(* CODESYS project GardenWatering.project
   Title: Garden Watering
   Version: 1.0
   Company: TK Automation
   Author: Toni Kucic

Project tree, tasks and I/O mapping:
  SoftPLC : CODESYS Control Win V3 x64, 3S - Smart Software Solutions GmbH, version 3.5.12.0
    application Application
      libraries: Standard, * (System); TkAutomationLib, 1.0 (TkAutomation); Util, * (System); Standard64, * (System); VisuDialogs, * (System)
      task VISU_TASK (cyclic, interval 50 ms, priority 31) calls VisuElems.Visu_Prg
      task xsim02 (cyclic, interval t#20ms, priority 2) calls xsim02
      task xc02_Task (cyclic, interval t#20ms, priority 1) calls xc02_GardenWatering, xc02_GardenWatering_Encoder
      FunctionalDescriptions/
        FD_GardenWatering
      image pool ImagePool
      FunctionBLocks/
        function block Servo [ST]
      IO/
        global variables xgv02
        Symbols
      Control/
        program xc02_GardenWatering [ST]
        program xc02_GardenWatering_Encoder [ST]
      Simulator/
        program xsim02 [ST]
      HMI/
        visualisation xv02_GardenWatering
  libraries: VisuSymbols, 3.5.10.0 (System)
  00000000-0000-0000-0000-000000000000|C:\Users\Toni\Google Drive\Projekti\PLC projekti\tkautomation school\Functional Descriptions\FD_GardenWatering.docx
  text list GlobalTextList
  5ce3da45-db07-42e7-a21c-a00fff4ed8f6|Car1.png
  5ce3da45-db07-42e7-a21c-a00fff4ed8f6|Projects\breaker1.jpg
  5ce3da45-db07-42e7-a21c-a00fff4ed8f6|Projects\breaker2.jpg
  5ce3da45-db07-42e7-a21c-a00fff4ed8f6|Projects\Ventilator1.jpg
  5ce3da45-db07-42e7-a21c-a00fff4ed8f6|Projects\Ventilator2.jpg
  5ce3da45-db07-42e7-a21c-a00fff4ed8f6|Projects\main-switchboard_1.jpg
  5ce3da45-db07-42e7-a21c-a00fff4ed8f6|Projects\breaker1.jpg
  5ce3da45-db07-42e7-a21c-a00fff4ed8f6|Projects\breaker2.jpg
  5ce3da45-db07-42e7-a21c-a00fff4ed8f6|Projects\cloud with rain.jpg
  5ce3da45-db07-42e7-a21c-a00fff4ed8f6|Car2.png
  text list System
  5ce3da45-db07-42e7-a21c-a00fff4ed8f6|Car3.png
  5ce3da45-db07-42e7-a21c-a00fff4ed8f6|Projects\Ventilator1small.jpg
  5ce3da45-db07-42e7-a21c-a00fff4ed8f6|Projects\Ventilator2small.jpg
  5ce3da45-db07-42e7-a21c-a00fff4ed8f6|Projects\igrasatasterima.JPG
  5ce3da45-db07-42e7-a21c-a00fff4ed8f6|Projects\empty-road-intersection-icon-cartoon-style-H67GFG.jpg
  5ce3da45-db07-42e7-a21c-a00fff4ed8f6|Projects\traffic_light_05.jpgsmall.jpg
  5ce3da45-db07-42e7-a21c-a00fff4ed8f6|Projects\breaker1.jpg
  5ce3da45-db07-42e7-a21c-a00fff4ed8f6|Projects\breaker2.jpg
  5ce3da45-db07-42e7-a21c-a00fff4ed8f6|C:\Users\Toni\Google Drive\Projekti\PLC projekti\Materijali\traffic_light_05.jpgsmall.jpg
  5ce3da45-db07-42e7-a21c-a00fff4ed8f6|boom.png
  5ce3da45-db07-42e7-a21c-a00fff4ed8f6|bottle_empty.png
  5ce3da45-db07-42e7-a21c-a00fff4ed8f6|bottle_broken.png
  5ce3da45-db07-42e7-a21c-a00fff4ed8f6|bottle_halffull.png
  5ce3da45-db07-42e7-a21c-a00fff4ed8f6|bottle_full.png
  5ce3da45-db07-42e7-a21c-a00fff4ed8f6|roller1.png
  5ce3da45-db07-42e7-a21c-a00fff4ed8f6|roller2.png
  5ce3da45-db07-42e7-a21c-a00fff4ed8f6|cranebackground.png
  5ce3da45-db07-42e7-a21c-a00fff4ed8f6|cranemover.png
  5ce3da45-db07-42e7-a21c-a00fff4ed8f6|hook.png
  5ce3da45-db07-42e7-a21c-a00fff4ed8f6|trafficlightsystem.jpg
  5ce3da45-db07-42e7-a21c-a00fff4ed8f6|Car4.png
*)

// SoftPLC/Application/IO/xgv02
{attribute 'qualified_only'}
VAR_GLOBAL
	
	//Configuration

	//Inputs
	HorizontalS1 : BOOL;
	HorizontalS2 : BOOL;
	VerticalS1 : BOOL;
	VerticalS2 : BOOL;
	
	//Data from encoder
	PositionX : REAL;
	PositionY : REAL;
	
	(* HMI *)
	HMIUp : BOOL;
	HMIDown : BOOL;
	HMIRight : BOOL;
	HMILeft : BOOL;
	HMIUpRight : BOOL;
	HMIUpLeft : BOOL;
	HMIDownRight : BOOL;
	HMIDownLeft : BOOL;
	HMICoorXCmd : REAL;
	HMICoorYCmd : REAL;
	HMIOpenWater : BOOL;
	Remote : BOOL;
	Reset : BOOL;
	
	//Outputs
	HorizontalRight : BOOL;
	HorizontalLeft : BOOL;
	VerticalUp: BOOL;
	VerticalDown : BOOL;
	OpenWaterValve : BOOL;
END_VAR

// SoftPLC/Application/Simulator/xsim02
PROGRAM xsim02
VAR
	CollisionDetector: CollisionDetection;
	FlowerDeathTimer: TON;
	vResetSIM: BOOL;
	vFlowers : ARRAY [0..59] OF DWORD := [60(16#FF73B98B)];
	i : INT;
vFlowersXY : ARRAY [0..59, 0..1] OF INT := [276,253,	381,253,	486,253,	591,253,	696,253,	801,253,	906,253,	1011,253,	1116,253,	1221,253,
												276,354,	381,354,	486,354,	591,354,	696,354,	801,354,	906,354,	1011,354,	1116,354,	1221,354,
												276,455,	381,455,	486,455,	591,455,	696,455,	801,455,	906,455,	1011,455,	1116,455,	1221,455,
												276,556,	381,556,	486,556,	591,556,	696,556,	801,556,	906,556,	1011,556,	1116,556,	1221,556,
												276,667,	381,667,	486,667,	591,667,	696,667,	801,667,	906,667,	1011,667,	1116,667,	1221,667,
												276,768,	381,768,	486,768,	591,768,	696,768,	801,768,	906,768,	1011,768,	1116,768,	1221,768]; (* Coordinates of flowers in format Flower0 -x,y *)

END_VAR

(* If the plaform covers the flower it will reset its color to initial *)
FOR i:=0 TO 59 BY 1 DO
	CollisionDetector(
		xcor1:= xgv02.PositionX, 
		ycor1:= xgv02.PositionY, 
		height1:= 10, 
		width1:= 10, 
		xcor2:= vFlowersXY[i,0], 
		ycor2:= vFlowersXY[i,1], 
		height2:= 70 , 
		width2:= 70);
	IF CollisionDetector.isCollision AND xgv02.OpenWaterValve THEN
		vFlowers[i] := 16#FF73B98B;
	END_IF
END_FOR

FlowerDeathTimer(IN:=TRUE, PT:=T#60S);
(* Flowers fade its color *)
IF FlowerDeathTimer.Q THEN
	FOR i:=0 TO 59 BY 1 DO
		IF vFlowers[i] > 16#0073B98B THEN
			vFlowers[i] := vFlowers[i] - 16#01000000;
		END_IF;
	END_FOR
	FlowerDeathTimer.IN := FALSE;
END_IF;

END_PROGRAM

// SoftPLC/Application/Control/xc02_GardenWatering
PROGRAM xc02_GardenWatering
VAR
	vFlowersXY : ARRAY [0..59, 0..1] OF INT := [276,253,	381,253,	486,253,	591,253,	696,253,	801,253,	906,253,	1011,253,	1116,253,	1221,253,
												276,354,	381,354,	486,354,	591,354,	696,354,	801,354,	906,354,	1011,354,	1116,354,	1221,354,
												276,455,	381,455,	486,455,	591,455,	696,455,	801,455,	906,455,	1011,455,	1116,455,	1221,455,
												276,556,	381,556,	486,556,	591,556,	696,556,	801,556,	906,556,	1011,556,	1116,556,	1221,556,
												276,667,	381,667,	486,667,	591,667,	696,667,	801,667,	906,667,	1011,667,	1116,667,	1221,667,
												276,768,	381,768,	486,768,	591,768,	696,768,	801,768,	906,768,	1011,768,	1116,768,	1221,768]; (* Coordinates of flowers in format Flower0 -x,y *)

	vManual: BOOL;
	vXCMD : REAL;
	vYCMD : REAL;
	i: INT;
	Watering: TON;
	ActuatorOverFlower : CollisionDetection;
END_VAR

(* Control from the graphics *)
IF NOT xgv02.Remote THEN
	xgv02.HorizontalLeft := xgv02.HMIDownLeft OR xgv02.HMILeft OR xgv02.HMIUpLeft;
	xgv02.HorizontalRight := xgv02.HMIDownRight OR xgv02.HMIRight OR xgv02.HMIUpRight;
	xgv02.VerticalUp := xgv02.HMIUpLeft OR xgv02.HMIUp OR xgv02.HMIUpRight;
	xgv02.VerticalDown := xgv02.HMIDownLeft OR xgv02.HMIDown OR xgv02.HMIDownRight;
	xgv02.OpenWaterValve := xgv02.HMIOpenWater;
END_IF;

(* Coordinate control *)
IF xgv02.Remote AND vManual THEN
	vXCMD := xgv02.HMICoorXCmd;
	vYCMD := xgv02.HMICoorYCmd;
ELSE
	xgv02.HMICoorXCmd := xgv02.PositionX;
	xgv02.HMICoorYCmd := xgv02.PositionY;
END_IF

(* Full automatic algorithm *)
IF xgv02.Remote AND NOT vManual THEN
	vXCMD := vFlowersXY[i,0]+ 30;
	vYCMD := vFlowersXY[i,1]+ 30;
	
	ActuatorOverFlower(
		xcor1:= xgv02.PositionX, 
		ycor1:= xgv02.PositionY, 
		height1:= 10, 
		width1:= 10, 
		xcor2:= vFlowersXY[i,0], 
		ycor2:= vFlowersXY[i,1], 
		height2:= 70, 
		width2:= 70);
		
	IF 	ActuatorOverFlower.isCollision THEN
		Watering(IN:=TRUE, PT:=T#3S);
		xgv02.OpenWaterValve := TRUE;
	END_IF;
	IF ActuatorOverFlower.isCollision AND Watering.Q THEN
		Watering(IN := FALSE);
		xgv02.OpenWaterValve:= FALSE;
		i:= i + 1;	
	END_IF
END_IF
IF i = 59 THEN
	i := 0;
END_IF

(* Actual motor movement section *)
IF xgv02.Remote THEN
	IF vXCMD > xgv02.PositionX - 2 THEN
		xgv02.HorizontalLeft := FALSE;
		xgv02.HorizontalRight := TRUE;
	ELSIF vXCMD < xgv02.PositionX + 2 THEN
		xgv02.HorizontalLeft := TRUE;
		xgv02.HorizontalRight := FALSE;
	ELSE
		xgv02.HorizontalLeft := FALSE;
		xgv02.HorizontalRight := FALSE;
	END_IF;
	
	IF vYCMD < xgv02.PositionY - 2THEN
		xgv02.VerticalUp := TRUE;
		xgv02.VerticalDown := FALSE;
	ELSIF vYCMD > xgv02.PositionY + 2 THEN
		xgv02.VerticalUp := FALSE;
		xgv02.VerticalDown := TRUE;
	ELSE
		xgv02.VerticalUp := FALSE;
		xgv02.VerticalDown := FALSE;
	END_IF;
END_IF;

END_PROGRAM

// SoftPLC/Application/Control/xc02_GardenWatering_Encoder
PROGRAM xc02_GardenWatering_Encoder
VAR
	HorizontalAxis: Servo;
	VerticalAxis: Servo;
	rtHIncrement : R_TRIG;
	rtHDecrement : R_TRIG;
	rtVIncrement : R_TRIG;
	rtVDecrement : R_TRIG;
	vHorizontalS1Old: BOOL;
	vHorizontalS2Old: BOOL;
	vVerticalS1Old: BOOL;
	vVerticalS2Old: BOOL;
	PositionCounterVerticalAxis: CTUD;
	vHorizontalPos: DINT;
	PositionCounterHorizontalAxis: CTUD;
	vVerticalPos: WORD;
	vPositionX: REAL;
	vPositionY: REAL;
	vHorizontalLimit: BOOL;
	vVerticalLimit: BOOL;
	vPlatformActualPosX : REAL;
	vPlatformActualPosY : REAL;
END_VAR

(* The actual servos that move the watering equipment *)
vHorizontalLimit := (vPositionX >= 940 AND NOT xgv02.HorizontalLeft)
				  OR (vPositionX <= 0 AND NOT xgv02.HorizontalRight);
vVerticalLimit := (vPositionY >= 500 AND NOT xgv02.VerticalUp)
			    OR (vPositionY <= 0 AND NOT xgv02.VerticalDown);

(* Maximum range - 940 steps *)
HorizontalAxis(
	CmdFwd:= xgv02.HorizontalRight AND NOT vHorizontalLimit, 
	CmdRev:= xgv02.HorizontalLeft AND NOT vHorizontalLimit, 
	PulseWidth:= T#0.1S , 
	S1=> xgv02.HorizontalS1, 
	S2=> xgv02.HorizontalS2);
	
(* Maximum range - 500 steps *)	
VerticalAxis(
	CmdFwd:= xgv02.VerticalDown AND NOT vVerticalLimit, 
	CmdRev:= xgv02.VerticalUp AND NOT vVerticalLimit, 
	PulseWidth:= T#0.1S , 
	S1=> xgv02.VerticalS1, 
	S2=> xgv02.VerticalS2);

IF xgv02.HorizontalS1 <> vHorizontalS1Old THEN
	IF xgv02.HorizontalS1 <> xgv02.HorizontalS2 THEN
		rtHIncrement(CLK:=TRUE);
	ELSE
		rtHDecrement(CLK:=TRUE);
	END_IF
ELSE
	rtHIncrement(CLK:=FALSE);
	rtHDecrement(CLK:=FALSE);
END_IF

IF xgv02.VerticalS1 <> vVerticalS1Old THEN
	IF xgv02.VerticalS1 <> xgv02.VerticalS2 THEN
		rtVIncrement(CLK:=TRUE);
	ELSE
		rtVDecrement(CLK:=TRUE);
	END_IF
ELSE
	rtVIncrement(CLK:=FALSE);
	rtVDecrement(CLK:=FALSE);
END_IF

PositionCounterHorizontalAxis(
	CU:= rtHIncrement.Q, 
	CD:= rtHDecrement.Q, 
	CV=> vHorizontalPos);

PositionCounterVerticalAxis(
	CU:= rtVIncrement.Q, 
	CD:= rtVDecrement.Q, 
	CV=> vVerticalPos);
	
(* Position of the system in the graphics*)
(* For every 1 pulses we move 5 px *)
vPositionX := (DINT_TO_REAL(vHorizontalPos)/ 1) * 5;
vPositionY := (DINT_TO_REAL(vVerticalPos)/ 1) * 5;
	
vHorizontalS1Old := xgv02.HorizontalS1;
vVerticalS1Old := xgv02.VerticalS1;
(* This is to counter the starting offset in the graphics *)
vPlatformActualPosX := 307 + vPositionX;
vPlatformActualPosY := 279 + vPositionY;

(* Send the platform position to other programs *)
xgv02.PositionX := vPlatformActualPosX;
xgv02.PositionY := vPlatformActualPosY;

END_PROGRAM

// SoftPLC/Application/FunctionBLocks/Servo
FUNCTION_BLOCK Servo
VAR_INPUT
	CmdFwd : BOOL := FALSE;
	CmdRev : BOOL := FALSE;
	PulseWidth : TIME := T#0.1S; (* Width of a pulse from the hall effect sensor when its above magnetic surface *)
END_VAR
VAR_OUTPUT
	S1 : BOOL := FALSE;
	S2 : BOOL := FALSE;
END_VAR
VAR
	tofS2 : TOF;
	tonS2 : TON;
	blink : BLINK;
	blinkOld: BOOL;
	vStartBlinker: BOOL;
END_VAR

vStartBlinker := (CmdFwd OR CmdRev) AND NOT (CmdFwd AND CmdRev);
Blink(ENABLE := vStartBlinker, TIMELOW:= PulseWidth, TIMEHIGH := PulseWidth);

tonS2(IN := blink.OUT, PT:=PulseWidth/2);
tofS2(IN := NOT tonS2.Q AND blinkOld, PT:=PulseWidth/2);
 
blinkOld := tonS2.Q;

IF CmdFwd THEN
	S1 := blink.OUT;
	S2 := tonS2.Q OR tofS2.Q;
ELSIF CmdRev THEN
	S1 := tonS2.Q OR tofS2.Q;
	S2 := blink.OUT;
END_IF

END_FUNCTION_BLOCK

// SoftPLC/Application/HMI/xv02_GardenWatering
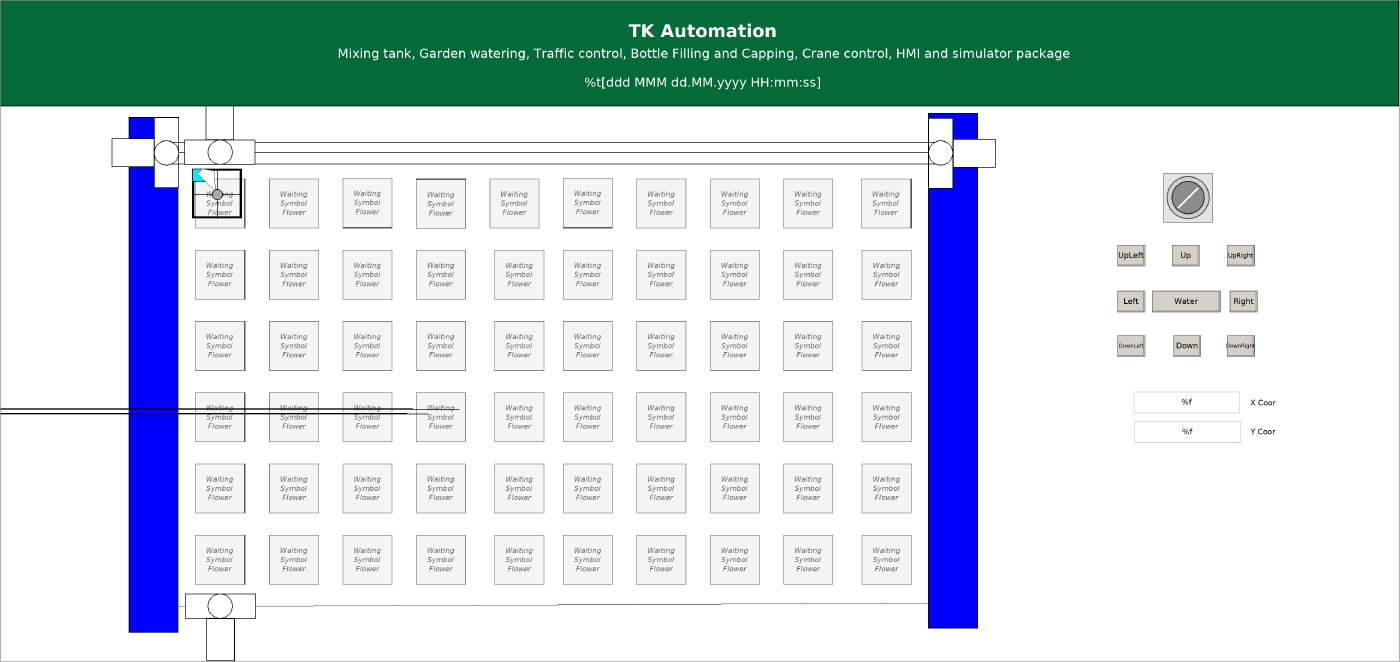
VISUALIZATION xv02_GardenWatering  // 1982x938
    RoundedRectangle (381,354 70x70), colour variable: xsim02.vFlowers[11]
    RoundedRectangle (485,354 70x70), colour variable: xsim02.vFlowers[12]
    RoundedRectangle (589,354 70x70), colour variable: xsim02.vFlowers[13]
    RoundedRectangle (700,354 70x70), colour variable: xsim02.vFlowers[14]
    RoundedRectangle (797,354 70x70), colour variable: xsim02.vFlowers[15]
    RoundedRectangle (901,354 70x70), colour variable: xsim02.vFlowers[16]
    RoundedRectangle (1005,354 70x70), colour variable: xsim02.vFlowers[17]
    RoundedRectangle (1109,354 70x70), colour variable: xsim02.vFlowers[18]
    RoundedRectangle (1220,354 70x70), colour variable: xsim02.vFlowers[19]
    RoundedRectangle (381,455 70x70), colour variable: xsim02.vFlowers[21]
    RoundedRectangle (485,455 70x70), colour variable: xsim02.vFlowers[22]
    RoundedRectangle (589,455 70x70), colour variable: xsim02.vFlowers[23]
    RoundedRectangle (700,455 70x70), colour variable: xsim02.vFlowers[24]
    RoundedRectangle (797,455 70x70), colour variable: xsim02.vFlowers[25]
    RoundedRectangle (901,455 70x70), colour variable: xsim02.vFlowers[26]
    RoundedRectangle (1005,455 70x70), colour variable: xsim02.vFlowers[27]
    RoundedRectangle (1109,455 70x70), colour variable: xsim02.vFlowers[28]
    RoundedRectangle (1220,455 70x70), colour variable: xsim02.vFlowers[29]
    RoundedRectangle (381,556 70x70), colour variable: xsim02.vFlowers[31]
    RoundedRectangle (485,556 70x70), colour variable: xsim02.vFlowers[32]
    RoundedRectangle (589,556 70x70), colour variable: xsim02.vFlowers[33]
    RoundedRectangle (700,556 70x70), colour variable: xsim02.vFlowers[34]
    RoundedRectangle (797,556 70x70), colour variable: xsim02.vFlowers[35]
    RoundedRectangle (901,556 70x70), colour variable: xsim02.vFlowers[36]
    RoundedRectangle (1005,556 70x70), colour variable: xsim02.vFlowers[37]
    RoundedRectangle (1109,556 70x70), colour variable: xsim02.vFlowers[38]
    RoundedRectangle (1220,556 70x70), colour variable: xsim02.vFlowers[39]
    RoundedRectangle (381,657 70x70), colour variable: xsim02.vFlowers[41]
    RoundedRectangle (485,657 70x70), colour variable: xsim02.vFlowers[42]
    RoundedRectangle (589,657 70x70), colour variable: xsim02.vFlowers[43]
    RoundedRectangle (700,657 70x70), colour variable: xsim02.vFlowers[44]
    RoundedRectangle (797,657 70x70), colour variable: xsim02.vFlowers[45]
    RoundedRectangle (901,657 70x70), colour variable: xsim02.vFlowers[46]
    RoundedRectangle (1005,657 70x70), colour variable: xsim02.vFlowers[47]
    RoundedRectangle (1109,657 70x70), colour variable: xsim02.vFlowers[48]
    RoundedRectangle (1220,657 70x70), colour variable: xsim02.vFlowers[49]
    RoundedRectangle (381,758 70x70), colour variable: xsim02.vFlowers[51]
    RoundedRectangle (485,758 70x70), colour variable: xsim02.vFlowers[52]
    RoundedRectangle (589,758 70x70), colour variable: xsim02.vFlowers[53]
    RoundedRectangle (700,758 70x70), colour variable: xsim02.vFlowers[54]
    RoundedRectangle (797,758 70x70), colour variable: xsim02.vFlowers[55]
    RoundedRectangle (901,758 70x70), colour variable: xsim02.vFlowers[56]
    RoundedRectangle (1005,758 70x70), colour variable: xsim02.vFlowers[57]
    RoundedRectangle (1109,758 70x70), colour variable: xsim02.vFlowers[58]
    RoundedRectangle (1220,758 70x70), colour variable: xsim02.vFlowers[59]
    Group (276,253 71x70)
        RoundedRectangle (1,0 70x70), colour variable: xsim02.vFlowers[0]
        WaitingSymbolFlower (0,0 70x70)
    Group (276,354 71x70)
        RoundedRectangle (1,0 70x70), colour variable: xsim02.vFlowers[10]
        WaitingSymbolFlower (0,0 70x70)
    Group (276,455 71x70)
        RoundedRectangle (1,0 70x70), colour variable: xsim02.vFlowers[20]
        WaitingSymbolFlower (0,0 70x70)
    Group (276,758 71x70)
        RoundedRectangle (1,0 70x70), colour variable: xsim02.vFlowers[50]
        WaitingSymbolFlower (0,0 70x70)
    Group (276,556 71x70)
        RoundedRectangle (1,0 70x70), colour variable: xsim02.vFlowers[30]
        WaitingSymbolFlower (0,0 70x70)
    Group (276,657 71x70)
        RoundedRectangle (1,0 70x70), colour variable: xsim02.vFlowers[40]
        WaitingSymbolFlower (0,0 70x70)
    Group (381,253 70x70)
        RoundedRectangle (0,0 70x70), colour variable: xsim02.vFlowers[1]
        WaitingSymbolFlower (0,0 70x70)
    WaitingSymbolFlower (381,354 70x70)
    WaitingSymbolFlower (381,455 70x70)
    WaitingSymbolFlower (381,758 70x70)
    WaitingSymbolFlower (381,556 70x70)
    WaitingSymbolFlower (381,657 70x70)
    Group (589,253 70x71)
        RoundedRectangle (0,0 70x70), colour variable: xsim02.vFlowers[2]
        WaitingSymbolFlower (0,1 70x70)
    WaitingSymbolFlower (485,354 70x70)
    WaitingSymbolFlower (485,455 70x70)
    WaitingSymbolFlower (485,758 70x70)
    WaitingSymbolFlower (485,556 70x70)
    WaitingSymbolFlower (485,657 70x70)
    Group (485,252 70x71)
        RoundedRectangle (0,1 70x70), colour variable: xsim02.vFlowers[3]
        WaitingSymbolFlower (0,0 70x70)
    WaitingSymbolFlower (589,354 70x70)
    WaitingSymbolFlower (589,455 70x70)
    WaitingSymbolFlower (589,758 70x70)
    WaitingSymbolFlower (589,556 70x70)
    WaitingSymbolFlower (589,657 70x70)
    Group (693,253 70x70)
        RoundedRectangle (0,0 70x70), colour variable: xsim02.vFlowers[4]
        WaitingSymbolFlower (0,0 70x70)
    WaitingSymbolFlower (700,354 70x70)
    WaitingSymbolFlower (700,455 70x70)
    WaitingSymbolFlower (700,758 70x70)
    WaitingSymbolFlower (700,556 70x70)
    WaitingSymbolFlower (700,657 70x70)
    Group (797,252 70x71)
        RoundedRectangle (0,1 70x70), colour variable: xsim02.vFlowers[5]
        WaitingSymbolFlower (0,0 70x70)
    WaitingSymbolFlower (797,354 70x70)
    WaitingSymbolFlower (797,455 70x70)
    WaitingSymbolFlower (797,758 70x70)
    WaitingSymbolFlower (797,556 70x70)
    WaitingSymbolFlower (797,657 70x70)
    Group (901,253 70x70)
        RoundedRectangle (0,0 70x70), colour variable: xsim02.vFlowers[6]
        WaitingSymbolFlower (0,0 70x70)
    WaitingSymbolFlower (901,354 70x70)
    WaitingSymbolFlower (901,455 70x70)
    WaitingSymbolFlower (901,758 70x70)
    WaitingSymbolFlower (901,556 70x70)
    WaitingSymbolFlower (901,657 70x70)
    Group (1005,253 70x70)
        RoundedRectangle (0,0 70x70), colour variable: xsim02.vFlowers[7]
        WaitingSymbolFlower (0,0 70x70)
    WaitingSymbolFlower (1005,354 70x70)
    WaitingSymbolFlower (1005,455 70x70)
    WaitingSymbolFlower (1005,758 70x70)
    WaitingSymbolFlower (1005,556 70x70)
    WaitingSymbolFlower (1005,657 70x70)
    Group (1109,253 70x70)
        RoundedRectangle (0,0 70x70), colour variable: xsim02.vFlowers[8]
        WaitingSymbolFlower (0,0 70x70)
    WaitingSymbolFlower (1109,354 70x70)
    WaitingSymbolFlower (1109,455 70x70)
    WaitingSymbolFlower (1109,758 70x70)
    WaitingSymbolFlower (1109,556 70x70)
    WaitingSymbolFlower (1109,657 70x70)
    Group (1219,253 71x70)
        RoundedRectangle (1,0 70x70), colour variable: xsim02.vFlowers[9]
        WaitingSymbolFlower (0,0 70x70)
    WaitingSymbolFlower (1220,354 70x70)
    WaitingSymbolFlower (1220,455 70x70)
    WaitingSymbolFlower (1220,758 70x70)
    WaitingSymbolFlower (1220,556 70x70)
    WaitingSymbolFlower (1220,657 70x70)
    Line (212,859) (1367,854)
    Rectangle (182,166 70x730)
    Rectangle (1314,160 70x730)
    Line (211,216) (1334,216)
    Rectangle (1314,167 35x100)
    RoundedRectangle (1349,197 60x40)
    Rectangle (218,166 35x100)
    RoundedRectangle (158,196 60x40)
    Line (230,201) (1336,201)
    Line (229,232) (1338,232)
    Ellipse (218,199 35x35)
    Line (-39,580) (650,580)
        p3560616238: xc02_GardenWatering_Encoder.vPositionX
    Line (-106,578) (584,578)
        p3560616238: xc02_GardenWatering_Encoder.vPositionX
    Line (-43,586) (606,586)
        p3560616238: xc02_GardenWatering_Encoder.vPositionX
    Line (-74,585) (576,585)
        p3560616238: xc02_GardenWatering_Encoder.vPositionX
    Group (261,138 100x95)
        p3560616238: xc02_GardenWatering_Encoder.vPositionX
        RoundedRectangle (30,0 40x60)
        Rectangle (0,60 100x35)
        Ellipse (33,60 35x35)
    Group (262,841 100x95)
        p3560616238: xc02_GardenWatering_Encoder.vPositionX
        Rectangle (0,0 100x35)
        RoundedRectangle (30,35 40x60)
        Ellipse (32,0 35x35)
    Ellipse (1314,199 35x35)
    Button (1659,347 39x30), "Up"
        tap xgv02.HMIUp
    Button (1661,475 39x30), "Down"
        tap xgv02.HMIDown
    Button (1741,412 39x30), "Right"
        tap xgv02.HMIRight
    Button (1582,412 39x30), "Left"
        tap xgv02.HMILeft
    Button (1737,347 39x30), "UpRight"
        tap xgv02.HMIUpRight
    Button (1582,347 39x30), "UpLeft"
        tap xgv02.HMIUpLeft
    Button (1582,475 39x30), "DownLeft"
        tap xgv02.HMIDownLeft
    Button (1737,475 39x30), "DownRight"
        tap xgv02.HMIDownRight
    Group (272,239 80x80)
        p3560616238: xc02_GardenWatering_Encoder.vPositionX
        p2738717112: xc02_GardenWatering_Encoder.vPositionY
        Rectangle (0,0 70x70)
        Line (0,36) (70,36)
        Line (35,0) (35,71)
        Rectangle (0,0 18x18)
        Polygon (7,7) (14,0) (31,3) (33,32) (30,29)
        Ellipse (28,29 15x15)
    RotarySwitch (1647,245 70x70), variable: xgv02.Remote, behaviour: TOGGLE, style: Switch-RotarySwitch-Gray
    Textfield (1605,555 150x30), "%f", text variable: xgv02.HMICoorXCmd
        OnMouseClick: write the text variable via Default
    Textfield (1606,597 150x30), "%f", text variable: xgv02.HMICoorYCmd
        OnMouseClick: write the text variable via Default
    Label (1763,556 50x30), "X Coor"
    Label (1763,597 50x30), "Y Coor"
    Button (1631,412 97x30), "Water"
        tap xgv02.HMIOpenWater
    Rectangle (0,0 1980x150)
    Label (839,27 312x33), "TK Automation"
    Label (244,61 1500x30), "Mixing tank, Garden watering, Traffic control, Bottle Filling and Capping, Crane control, HMI and simulator package"
    Rectangle (703,102 584x30), "%t[ddd MMM dd.MM.yyyy HH:mm:ss]"
END_VISUALIZATION

(* text list System (id | default)
  Apr | Apr
  April | April
  Aug | Aug
  August | August
  Dec | Dec
  December | December
  Feb | Feb
  February | February
  Fri | Fri
  Friday | Friday
  Jan | Jan
  January | January
  Jul | Jul
  July | July
  Jun | Jun
  June | June
  Mar | Mar
  March | March
  May | May
  May_3Letter | May
  Mon | Mon
  Monday | Monday
  Nov | Nov
  November | November
  Oct | Oct
  October | October
  Sat | Sat
  Saturday | Saturday
  Sep | Sep
  September | September
  Sun | Sun
  Sunday | Sunday
  Thu | Thu
  Thursday | Thursday
  Tue | Tue
  Tuesday | Tuesday
  Wed | Wed
  Wednesday | Wednesday
   |  *)
